FUNCTION_BLOCK FB_ROS2Connector EXTENDS FB_Base
VAR_INPUT
END_VAR
VAR_OUTPUT
END_VAR
VAR
END_VAR

CYCLIC_BASE();
HeartBeat();

{error 'Add method implementation or delete method to use base implementation'}
METHOD Activate : BOOL
END_METHOD

{error 'Add method implementation or delete method to use base implementation'}
METHOD Cleanup : BOOL
END_METHOD

{error 'Add method implementation or delete method to use base implementation'}
METHOD Configure : BOOL
END_METHOD

{error 'Add method implementation or delete method to use base implementation'}
METHOD Deactivate : BOOL
END_METHOD

{error 'Add method implementation or delete method to use base implementation'}
METHOD Destroy : BOOL
END_METHOD

{error 'Add method implementation or delete method to use base implementation'}
METHOD Shutdown : BOOL
END_METHOD

END_FUNCTION_BLOCK

(* stored: Version 1.1.0.1, ProductVersion 3.1.4026.18
   POU FB_ROS2Connector: Id {6a96c8c7-52cd-4751-affe-1665f30e203a}, SpecialFunc None
   Method Activate: Id {4246cd57-a8f1-4e05-80bb-46f1fc323209}
   Method Cleanup: Id {c09ff638-6fd3-453b-93c9-c293dde25a61}
   Method Configure: Id {58e52956-5985-4e99-8dea-09275ea2b32d}
   Method Deactivate: Id {9df0ddb3-f8f1-4521-97b6-96f891630978}
   Method Destroy: Id {37571124-ec1b-4c2d-afdc-8e3d36434ad3}
   Method Shutdown: Id {dbbf2126-71c3-4df2-907f-e50c0a4e32b5} *)
